ABB RAPID module: MainModule.mod

MODULE MainModule
	CONST robtarget pHome:=[[507.90,-6.43,715.02],[0.697685,-0.00154316,0.716328,-0.0103435],[-1,-1,-1,0],[9E+09,9E+09,9E+09,9E+09,9E+09,9E+09]];
	CONST robtarget conv:=[[-49.18,-617.16,499.98],[0.309443,0.549198,0.646739,-0.429365],[-2,-1,-1,0],[9E+09,9E+09,9E+09,9E+09,9E+09,9E+09]];
	CONST robtarget man:=[[635.90,42.30,481.74],[0.518931,-0.131239,0.843441,-0.0457607],[0,-1,-1,0],[9E+09,9E+09,9E+09,9E+09,9E+09,9E+09]];
	CONST robtarget oven:=[[-400.60,632.71,501.69],[0.350259,-0.742904,0.298477,0.486132],[1,-1,-1,0],[9E+09,9E+09,9E+09,9E+09,9E+09,9E+09]];
	PROC main()
		MoveL [[-400.60,632.72,501.69],[0.35026,-0.742905,0.298477,0.48613],[1,-1,-1,0],[9E+09,9E+09,9E+09,9E+09,9E+09,9E+09]], v1000, z50, tool0;
	ENDPROC
ENDMODULE
